{attribute 'linkalways'} 
{attribute 'no_explicit_call' := 'This FB is a CLASS and must be accessed using methods or properties'}
{attribute 'enable_dynamic_creation'}
FUNCTION_BLOCK Node_F_VN_FindTemplateWalsh EXTENDS VisionNode
VAR
    ipSrcImage : _ITcVnImage;
    ipTemplateImage : _ITcVnImage;
	ipMatches : _ITcVnContainer;
	fMatchThreshold : _REAL(0.1);
	nProjections : _UDINT(10);
    hrPrev : _HRESULT(S_OK);
	hresult : _HRESULT(S_OK);
END_VAR

METHOD PUBLIC  Clone : I_Node
VAR
	pNode : POINTER TO Node_F_VN_FindTemplateWalsh;
END_VAR
pNode := __NEW(Node_F_VN_FindTemplateWalsh);
Clone := pNode^;
END_METHOD

METHOD FB_init : BOOL
VAR_INPUT
	bInitRetains : BOOL; // if TRUE, the retain variables are initialized (warm start / cold start)
	bInCopyCode : BOOL;  // if TRUE, the instance afterwards gets moved into the copy code (online change)
END_VAR
AddInput('ipSrcImage', ipSrcImage);
AddInput('ipTemplateImage', ipTemplateImage);
AddInput('fMatchThreshold', fMatchThreshold);
AddInput('nProjections', nProjections);
AddInput('hrPrev', hrPrev);
AddOutput('ipMatches', ipMatches);
AddOutput('hresult',hresult);
END_METHOD

METHOD PROTECTED OnExecute
hresult.Value := F_VN_FindTemplateWalsh(
    ipSrcImage := ipSrcImage.Value,
    ipTemplateImage := ipTemplateImage.Value,
	ipMatches := ipMatches.Value,
	fMatchThreshold := fMatchThreshold.Value,
	nProjections := nProjections.Value,
	hrPrev:= hrPrev.Value);
END_METHOD

METHOD PUBLIC PreExecutionCheck
VAR_INPUT
	Check : I_PreExecutionChecks;
END_VAR
Check.IsTrue(ipSrcImage.IsValid, 'ipSrcImage must contain an image');
Check.IsTrue(ipSrcImage.IsPixelDepth(8), 'ipSrcImage must be 8 or 32 bit pixel depth');
Check.IsTrue((ipSrcImage.HasChannelCount(1) OR ipSrcImage.HasChannelCount(3)), 'ipSrcImage must contain 1 or 3 channels');

Check.IsTrue((fMatchThreshold.Value >= 0 AND fMatchThreshold.Value <= 1), 'Threshold must be between 0..1, 1.0 would be a perfect match');

Check.IsTrue(ipTemplateImage.IsValid, 'ipTemplateImage must contain an image');
Check.IsTrue(ImagesHaveMatchingPixelFormats(ipSrcImage.Value, ipTemplateImage.Value), 'ipTemplateImage must have same pixel depth as ipSrcImage');
Check.IsTrue(ImagesHaveMatchingChannels(ipSrcImage.Value, ipTemplateImage.Value), 'ipTemplateImage must have same amount of channels as ipSrcImage');
Check.IsTrue(IsTemplateImageSmallerThanSourceImage(ipSrcImage.Value, ipTemplateImage.Value), 'ipTemplateImage must be smaller than ipSrcImage');
END_METHOD

END_FUNCTION_BLOCK

(* stored: Version 1.1.0.1, ProductVersion 3.1.4026.13
   POU Node_F_VN_FindTemplateWalsh: Id {35903528-f141-0df4-29ad-cfcc13091666}, SpecialFunc None
   Folder Constructor: Id {ea25716f-8241-0b94-38b7-22226db3b25d}
   Method Clone: Id {7dfb6b49-1b86-081b-2734-2a2cadf25abe}
   Method FB_init: Id {961ce5b2-2f0d-0b78-2f14-f365f06e9334}
   Method OnExecute: Id {ea41db5c-5292-0415-397a-11443bda48d7}
   Method PreExecutionCheck: Id {0a2519c7-6f27-0dc8-36dc-3aa7b504cd6c} *)
